
// ===== library types =====

// folder: LIOLink

TYPE "LIOLink_typeDiagnostics"
   STRUCT
      status : Word;   // Status of the Block or error identification when error occurred
      subfunctionStatus : DWord;   // Status or return value of called FB's, FCs and system blocks
      stateNumber : DInt;   // State in the state machine of the block where the error occurred
   END_STRUCT;
END_TYPE

// folder: iJaw

TYPE "UDT_iJawDataRcv"
   STRUCT
      Gauge1 : Word;   // ADC Eingang der Sensorrohdaten (min.: 0 max.: 4096)
      Gauge2 : Word;   // ADC Eingang der Sensorrohdaten (min.: 0 max.: 4096)
      Battery : Byte;   // Rohsignal aktuelle Batteriespannung (min.: 0 .. max.: 157) [V]
      Temperature : Byte;   // Rohsignal Temperatursensor (min.: -40 .. max.: 125) [°C]
      GyroXaxis : Byte;   // Rohsignal Beschleunigungssensor X (min.: -128 .. max.: 127) [g]
      GyroYaxis : Byte;   // Rohsignal Beschleunigungssensor Y (min.: -128 .. max.: 127) [g]
      GyroZaxis : Byte;   // Rohsignal Beschleunigungssensor Z (min.: -128 .. max.: 127) [g]
      Warning : Byte;   // Warnungs-/Fehlercode (Bit0:= Klemmkraft überschritten; Bit1:= Klemmkraft unters
      Force1 : Word;   // Spannkraft Kanal 1 (min.: 0 .. max.: 65,535) [N]
      Force2 : Word;   // Spannkraft Kanal 2 (min.: 0 .. max.: 65,535) [N]
      Reserve1431 : Array[14..31] of Byte;   // Reserve
   END_STRUCT;
END_TYPE

TYPE "UDT_iJawDataSend"
   STRUCT
      nRotSpeedSpindleAct : Int;   // actual rotational speed of the spindle
      pHydCylChamber1Act : Byte;   // actual hydraulic pressure in actuating cylinder chamber for outer clamping
      pHydCylChamber2Act : Byte;   // actual hydraulic pressure in actuating cylinder chamber for outer clamping
      AHydCylChamber1Act : Byte;   // hydraulic area of cylinder chamber for outer clamping
      AHydCylChamber2Act : Byte;   // hydraulic area of cylinder chamber for outer clamping
      Reserve0631 : Array[6..31] of Byte;   // Reserve
   END_STRUCT;
END_TYPE

TYPE "UDT_iJawDataSendUser"
   STRUCT
      xRelCmdSysMode : Bool;   // Trigger send Command change System Mode (see bMode)
      xRelCmdShotOff : Bool;   // Triggr send Command Shut Off
      xRelCmdTara : Bool;   // Trigger send Command Tara
      xReserve1 : Bool;   // Res
      xReserve2 : Bool;   // Res
      xReserve3 : Bool;   // Res
      xReserve4 : Bool;   // Res
      xReserve5 : Bool;   // Res
      bMode : Byte;   // Select Mode (0x1 = continuous mode; 0x2 = state dependent mode
      nRotSpeedSpindleAct : Int;   // actual rotational speed of the spindle
      pHydCylChamber1Act : Byte;   // actual hydraulic pressure in actuating cylinder chamber for outer clamping
      pHydCylChamber2Act : Byte;   // actual hydraulic pressure in actuating cylinder chamber for outer clamping
      AHydCylChamber1Act : Byte;   // hydraulic area of cylinder chamber for outer clamping
      AHydCylChamber2Act : Byte;   // hydraulic area of cylinder chamber for outer clamping
   END_STRUCT;
END_TYPE

TYPE "UDT_iJawDataRcvUser"
   STRUCT
      Gauge1 : UInt;   // ADC Eingang der Sensorrohdaten (min.: 0 max.: 4096)
      Gauge2 : UInt;   // ADC Eingang der Sensorrohdaten (min.: 0 max.: 4096)
      Battery : USInt;   // Rohsignal aktuelle Batteriespannung (min.: 0 .. max.: 157) [V]
      Temperature : SInt;   // Rohsignal Temperatursensor (min.: -40 .. max.: 125) [°C]
      GyroXaxis : SInt;   // Rohsignal Beschleunigungssensor X (min.: -128 .. max.: 127) [g]
      GyroYaxis : SInt;   // Rohsignal Beschleunigungssensor Y (min.: -128 .. max.: 127) [g]
      GyroZaxis : SInt;   // Rohsignal Beschleunigungssensor Z (min.: -128 .. max.: 127) [g]
      Warning : Byte;   // Warnungs-/Fehlercode (Bit0:= Klemmkraft überschritten; Bit1:= Klemmkraft unters
      Force1 : UInt;   // Spannkraft Kanal 1 (min.: 0 .. max.: 65,535) [N]
      Force2 : UInt;   // Spannkraft Kanal 2 (min.: 0 .. max.: 65,535) [N]
      Reserve1431 : Array[14..31] of Byte;   // Reserve
   END_STRUCT;
END_TYPE

// folder: LIOLink/S7-1200/1500/Base blocks

FUNCTION_BLOCK "LIOLink_Device"   // FB50004, SCL
TITLE = LIOLink_Device / LIOLINK_DEVICE
{ S7_Optimized_Access := 'TRUE' }
AUTHOR : SIOS
FAMILY : LIOLink
VERSION : 4.0
// Acyclically reads or writes data records from and to IO-Link devices / Funktionsbaustein zum Lesen und Schreiben von azyklischen Daten auf Geräten mit IO-Link, die auf SIMATIC S7-Steuerungen verwendet werden. (früher IO_LINK_CALL)
   VAR_INPUT
      execute : Bool;   // Request to execute function / Anforderung zum Ausführen der Funktion
      hwID : HW_IO;   // Hardware identifier of IO-Link master module or first sub module / Hardware-Kennung des IO-Link-Mastermoduls (Submodul für ET 200eco PN)
      cap : Int;   // Client Access Point (CAP) 0xB400 or 0x00E3 (227) / Client Access Point (CAP); 0xB400 für ET 200eco PN, CM 8x IO-Link, sonst 0xE003 (227)
      readWrite : Bool;   // FALSE: read-mode, TRUE: write-mode / FALSE: lesen, TRUE: schreiben
      port : Int;   // Port on IO-Link master module / Port am IO-Link-Master-Modul
      index : Int;   // Address parameter index (IO-Link device); 0..32767: IOL-D; 65535: port functions / Adressparameterindex (IO-Link Device); 0..32767: IOL-D; 65535: Portfunktionen
      subindex : Int;   // Address parameter subindex (IO-Link device); 0: full record; 1-255: single parameter / Adressparameter Subindex (IO-Link Device); 0: vollständige Aufzeichnung; 1-255: Einzelparameter
      writeLen : Int;   // Length of writing data (net data); 1..232 / Länge der Schreibdaten (Nettodaten); 1..232
      timeout : Time := T#20S;   // Time after which the request is aborted / Zeit, nach der die Anfrage abgebrochen wird
      pollingPeriod : Time := T#100MS;   // Time period of polling
   END_VAR
   VAR_OUTPUT
      done : Bool;   // TRUE: FB processing successfully completed / TRUE: FB-Bearbeitung erfolgreich abgeschlossen
      busy : Bool;   // TRUE: FB is active and new output values can be expected. / TRUE: FB ist aktiv und neue Ausgangswerte sind zu erwarten.
      error : Bool;   // FALSE: No error / TRUE: An error occurred during the execution of the FB. / FALSE: Kein Fehler / TRUE: Bei der Ausführung des FB ist ein Fehler aufgetreten.
      status : Word := 16#7000;   // 16#0000-16#7FFF: Status of the FB / 16#8000-16#FFFF: Error identification (see following table) / 16#0000-16#7FFF: Status des FB / 16#8000-16#FFFF: Fehleridentifikation (siehe folgende Tabelle)
      diagnostics : "LIOLink_typeDiagnostics";   // Diagnostics information of FB / Diagnoseinformationen der FB
      readLen : Int;   // Length of read data record (number of bytes) / Länge des gelesenen Datensatzes (Anzahl Bytes)
   END_VAR
   VAR_IN_OUT
      record : Array[*] of Byte;   // Data area for reading/writing data (max. 232 byte) / Datenbereich zum Lesen/Schreiben von Daten (max. 232 Byte)
   END_VAR
   VAR
      statExecuteOld : Bool;   // Old value of 'execute' input for edge detection / Alter Wert des 'Execute'-Eingangs für Flankenerkennung
      statDone : Bool;   // Static value for output 'done' / Statischer Wert für Ausgang 'done'
      statBusy : Bool;   // Static value for output 'busy' / Statischer Wert für Ausgang 'besetzt'
      statError : Bool;   // Static value for output 'error' / Statischer Wert für Ausgang 'error'
      statStatus : Word := 16#7000;   // Static value for output 'status' / Statischer Wert für Ausgang 'Status'
      statPollingPeriod : Time := T#100MS;   // Static value for input 'pollingPeriod'
      statHwID : HW_IO;   // Static value for input 'hwID' / Statischer Wert für Eingang 'hwID'
      statHwIDprevious : HW_IO;   // Static value for input 'hwID' from the previous execute / Statischer Wert für Eingang 'hwID'
      statReadWrite : Bool;   // Static value for input 'readWrite' / Stativwert für Eingabe 'readWrite'
      statCap : UInt;   // Static value for input 'cap' / Statischer Wert für Eingabe 'cap'
      statTimeout : Time;   // Static value for input 'timeout' / Statischer Wert für Eingang 'timeout'
      statLen : UInt;   // Length of data to be written to device / Länge der Daten, die auf das Gerät geschrieben werden sollen
      statSubfunctionStatus : DWord;   // Status of WRREC/RDREC or error code from IO-Link Master (%W1: IO-Link Master error, %W0: ISDU error) / Status von WRREC/RDREC oder Fehlercode vom IO-Link-Master (%W1: IO-Link-Master-Fehler, %W0: ISDU-Fehler)
      statFBErrorState : DInt;   // State in the state machine of the block where the error occurred / Zustand in der Zustandsmaschine des Blocks, in dem der Fehler aufgetreten ist
      statFBState : DInt := 0;   // State in the state machine of the FB / Zustand in der Zustandsmaschine der FB
      statEmptyDiagnostics : "LIOLink_typeDiagnostics";   // Empty diagnostics information (for initialization purposes only) / Leere Diagnoseinformationen (nur für Initialisierungszwecke)
      instRdRec : RDREC;   // System function "read data record" / Systemfunktion "Datensatz lesen"
      instWrRec : WRREC;   // System function "write data record" / Systemfunktion "Datensatz schreiben"
      instPoll : TP_TIME;   // poll rate read data record / Abfragerate Datensatz lesen
      instMonitor : TON_TIME;   // request monitoring time / Überwachungszeit anfordern
      statRead : Struct   // data area for reading data / Datenbereich zum Lesen von Daten
         header : Struct   // Header
            call : Struct   // header for read/write data record / Header für Datensatz lesen/schreiben
               extFunctionNum : Byte := 16#08;   // extended function number (fix coded 08h) / erweiterte Funktionsnummer (fix codiert 08h)
               port : Byte;   // variable port (user interface) 0...255 / variabler Port (Benutzeroberfläche) 0...255
               fiIndex : Word := 16#FE4A;   // FI index (fix coded 65098) / FI-Index (fix codiert 65098)
            END_STRUCT;
            iolHeader : Struct   // header for IO-Link / Header für IO-Link
               control : Byte;   // RD_WR = 0 = read = Control:=0x03 / / RD_WR = 1 = write = Control:=0x02 / RD_WR = 0 = lesen = Steuerung:=0x03 / / RD_WR = 1 = schreiben = Steuerung:=0x02
               indexHighByte : Byte;   // index of data record 0…32767 (high byte) / Index des Datensatzes 0…32767 (High Byte)
               indexLowByte : Byte;   // index of data record 0…32767 (low byte) / Index des Datensatzes 0…32767 (Low Byte)
               subindex : Byte;   // subindex for data record 0...255 / Subindex für Datensatz 0...255
            END_STRUCT;
         END_STRUCT;
         data : Array[0..231] of Byte;   // Data
      END_STRUCT;
      statWrite : Struct   // data area for writing data / Datenbereich zum Schreiben von Daten
         header : Struct   // Header
            call : Struct   // header for read/write data record / Header für Datensatz lesen/schreiben
               extFunctionNum : Byte := 16#08;   // extended function number (fix coded 08h) / erweiterte Funktionsnummer (fix codiert 08h)
               port : Byte;   // variable port (user interface) 0...255 / variabler Port (Benutzeroberfläche) 0...255
               fiIndex : Word := 16#FE4A;   // FI index (fix coded 65098) / FI-Index (fix codiert 65098)
            END_STRUCT;
            iolHeader : Struct   // header für IO-Link / Header für IO-Link
               control : Byte;   // RD_WR = 0 = read = Control:=0x03 / / RD_WR = 1 = write = Control:=0x02 / RD_WR = 0 = lesen = Steuerung:=0x03 / / RD_WR = 1 = schreiben = Steuerung:=0x02
               indexHighByte : Byte;   // index of data record 0…32767 (high byte) / Index des Datensatzes 0…32767 (High Byte)
               indexLowByte : Byte;   // index of data record 0…32767 (low byte) / Index des Datensatzes 0…32767 (Low Byte)
               subindex : Byte;   // subindex for data record 0...255 / Subindex für Datensatz 0...255
            END_STRUCT;
         END_STRUCT;
         data : Array[0..231] of Byte;   // Data
      END_STRUCT;
   END_VAR
   VAR_TEMP
      tempExecute : Bool;   // Temporary value for input 'execute' / Temporärer Wert für Eingabe 'execute'
      tempHwID : HW_IO;   // Temporary value for input 'hwID'
      tempPort : Int;   // Temporary value for input 'port'
      tempIndex : Int;   // Temporary value for input 'index'
      tempSubindex : Int;   // Temporary value for input 'subindex'
      tempIndexCounter : DInt;   // run tag for counting loops / Run-Tag für Zählschleifen
   END_VAR
   VAR CONSTANT
      MODE_READ : Bool := FALSE;   // Mode to read data / Modus zum Lesen von Daten
      MODE_WRITE : Bool := TRUE;   // Mode to write data / Modus zum Schreiben von Daten
      MAX_PORT : USInt := 63;   // Max. possible port / max. möglichen Hafen
      MAX_INDEX : UInt := 32767;   // Max. possible index / max. möglicher Index
      INDEX_PORT_FUNC : UInt := 65535;   // Index to address port functions / Index zum Adressieren von Portfunktionen
      MAX_SUBINDEX : USInt := 255;   // Max. possible subindex / max. möglicher Subindex
      MAX_DATA : USInt := 232;   // Max. size of data to be transferred / max. Größe der zu übertragenden Daten
      UPPER_LIMIT : DInt := 231;   // Upper limit of data to be transferred / Obergrenze der zu übertragenden Daten
      FB_STATE_NO_PROCESSING : DInt := 0;   // FB state: No processing / FB-Zustand: Keine Verarbeitung
      FB_STATE_WRITE : DInt := 1;   // FB state: Write data record / Datensatz schreiben
      FB_STATE_POLL : DInt := 2;   // FB state: Wait and poll for response / warten und auf Antwort abfragen
      FB_STATE_READ_CAP : DInt := 3;   // FB state: Read cap / CAP lesen
      IOL_HEADER : UInt := 65098;   // Header IO-Link / Kopfzeile IO-Link
      LEN_HEADER : USInt := 8;   // Length of header / Länge des Headers
      CONTROL_WRITE : Byte := 16#02;   // Write data record / Datensatz schreiben
      CONTROL_READ : Byte := 16#03;   // Read data record / Datensatz lesen
      STATUS_EXECUTION_FINISHED : Word := 16#0000;   // Execution finished without errors / Ausführung ohne Fehler beendet
      STATUS_NO_CALL : Word := 16#7000;   // No job being currently processed / Derzeit wird kein Auftrag bearbeitet
      STATUS_FIRST_CALL : Word := 16#7001;   // First call after incoming new job (rising edge 'execute') / Erster Aufruf nach eingehendem neuen Auftrag (steigende Flanke 'execute')
      STATUS_SUBSEQUENT_CALL : Word := 16#7002;   // Subsequent call during active processing without further details / Nachfolgender Aufruf während aktiver Bearbeitung ohne weitere Angaben
      SUB_STATUS_NO_ERROR : Word := 16#0000;   // No error occured in subfunction call / Fehler: falscher Port
      ERR_WRONG_PORT : Word := 16#8201;   // Error: wrong port / Fehler: falscher Index
      ERR_WRONG_INDEX : Word := 16#8202;   // Error: wrong index / Fehler: falscher Subindex
      ERR_WRONG_SUBINDEX : Word := 16#8203;   // Error: wrong subindex / Fehler: falsche Länge für Datensatz schreiben
      ERR_WRONG_LENGTH : Word := 16#8205;   // Error: wrong length for write data record / Fehler: IO-Link-Master hat Fehlercode zurückgegeben, siehe "Diagnose"
      ERR_IO_LINK : Word := 16#8401;   // Error: IO-Link master returned error code, see "diagnostics" / Fehler: Gelesener Datensatz stimmt nicht mit Anfrage überein
      ERR_INCONSISTENT_DATA : Word := 16#8402;   // Error: Read data record doesn't match request / Fehler: Zeitüberschreitung bei Anforderung
      ERR_REQUEST_TIMEOUT : Word := 16#8403;   // Error: Request timed out / Fehler: Aufgrund eines undefinierten Zustands in der Zustandsmaschine
      ERR_UNDEFINED_STATE : Word := 16#8600;   // Error: due to an undefined state in state machine / Fehler: Aufgrund eines undefinierten Zustands in der Zustandsmaschine
      ERR_WRREC : Word := 16#8601;   // Error: WRREC encountered an error, see "diagnostics" / Fehler: WRREC hat einen Fehler festgestellt, siehe "Diagnose"
      ERR_RDREC : Word := 16#8602;   // Error: RDREC encountered an error, see "diagnostics" / Fehler: RDREC hat einen Fehler festgestellt, siehe "Diagnose"
      STATUS_MASK : DWord := 16#00FF_FF00;   // Mask to filter error codes / Maske zum Filtern von Fehlercodes
      STATUS_RESOURCE_BUSY : DWord := 16#0080_C200;   // Status from WRREC/RDREC: Resource is busy / Status von WRREC/RDREC: Ressource ist beschäftigt
      INDEX_CAP_IOLINK : Word := 16#B000;   // Index of the data record for IOLM_Info. Only IO-Link-Masters with CAP=16#B000 support this call. / Index des Datensatzes für IOLM_Info. Nur IO-Link-Master mit CAP=16#B000 unterstützen diesen Aufruf.
      CAP_LEGACY : Word := 16#00E3;   // Siemens (old) Standard CAP: 227 / Siemens (alt) Standard CAP: 227
      CAP_STANDARD : Word := 16#B400;   // IO-Link Standard CAP: 16#B400 / IO-Link-Standard-CAP: 16#B400
      STATUS_RDREC_VALID : Byte := 16#00;   // Status Code of RDREC in cased of no error occurs
      BITMASK_ERR_RDREC_B3 : Byte := 16#DE;   // Status Code of RDREC in case of an error when reading a data record
      BITMASK_ERR_RDREC_B2 : Byte := 16#80;   // Status Code of RDREC in case of an error when reading a data record - Error according to IEC 61158-6
      BITMASK_ERR_RDREC_B1 : Byte := 16#B0;   // Status Code of RDREC in case of an error when reading a data record - invalid index (cap)
   END_VAR
BEGIN
   REGION BLOCK INFO HEADER
       //===============================================================================
       // Siemens / (c)Copyright 2023
       //-------------------------------------------------------------------------------
       // Title:            LIOLink_Device
       // Function:         Acyclically reads or writes data records from and to IO-Link devices
       // Library:          LIOLink
       // Author:           Siemens Industry Online Support
       // Tested with:      CPU 1513-1 PN FW 2.8
       // Engineering:      TIA Portal V16
       // Restrictions:     S7-1200/1500
       // Requirements:     --
       //-------------------------------------------------------------------------------
       // Change log table:
       // Version  | Date       | Expert in charge       | Changes applied
       //----------|------------|------------------------|------------------------------
       // 02.00.00 | 30.09.2013 | Online Support         | First release for TIA Portal V12 SP1 as IO_LINK_CALL
       // 02.01.00 | 14.03.2014 | Online Support         | Upgrade to TIA Portal V13
       //                                                | Upgrade of system function 'WRREC' from V1.0 to V1.1
       // 03.00.00 | 28.02.2015 | SUP Applications       | Upgrade to TIA Portal V13 SP1
       //                                                | Renamed FB to IO_LINK_DEVICE 
       // 03.01.00 | 15.09.2015 | SUP Applications       | Change of #IOL_INDEX AND #Port lower boundry to 0 and improved behaviour when called in cyclic OBs with > 100 ms
       // 04.00.00 | 01.09.2020 | Online Support         | Implemented Programming styleguide for S7-1200/1500 and PLCopen
       //                                                | Renamed FB to LIOLink_Device 
       // 05.00.00 | 28.02.2023 | SUP SPH                | Added Polling Time as predefined input
       //                                                | #record is changed to a variable array (Array[*])
       //                                                | Changed CAP as predefined variable, added functionality to automatically find CAP of IO-Link-Masters from SIEMENS                                               
       //===============================================================================
   END_REGION

   REGION TRIGGERING
       #tempExecute := #execute; // Work with temporary value / create process image

       IF (#tempExecute = TRUE) AND (#statExecuteOld = FALSE) // Check if FB is triggered
           AND (#statStatus = #STATUS_NO_CALL)
       THEN
           REGION Initialize data
               // First call; initialize FB
               #statDone := FALSE;
               #statBusy := TRUE;
               #statError := FALSE;
               #statStatus := #STATUS_FIRST_CALL;
               #statSubfunctionStatus := #SUB_STATUS_NO_ERROR;
               #statFBErrorState := 0;
               #diagnostics := #statEmptyDiagnostics;
               #readLen := 0;

               // Initialize data area
               #statRead.header."call"."port" := 16#0;
               #statRead.header.iolHeader.indexLowByte := 16#0;
               #statRead.header.iolHeader.indexHighByte := 16#0;
               #statRead.header.iolHeader.subindex := 16#0;
               #tempIndexCounter := 0; // initialize loop counter      
               FOR #tempIndexCounter := 0 TO #UPPER_LIMIT DO
                   #statWrite.data[#tempIndexCounter] := 16#0;
                   #statRead.data[#tempIndexCounter] := 16#0;
               END_FOR;
           END_REGION

           REGION Save inputs
               // Copy input variables to temporary variables
               #tempHwID := #hwID;
               #statReadWrite := #readWrite;
               #statTimeout := #timeout;
               #statPollingPeriod := #pollingPeriod;
               #tempPort := #port;
               #tempIndex := #index;
               #tempSubindex := #subindex;
           END_REGION

           REGION Build header
               // setup call header
               #statWrite.header."call"."port" := INT_TO_BYTE(#tempPort);

               // setup IOL header 
               #statWrite.header.iolHeader.indexLowByte := INT_TO_BYTE(#tempIndex);
               #statWrite.header.iolHeader.indexHighByte := INT_TO_BYTE(SHR(IN := #tempIndex, N := 8));
               #statWrite.header.iolHeader.subindex := INT_TO_BYTE(#tempSubindex);

               // BODY (data max. 232 Byte, Array 0..231 of Byte) 
               IF #statReadWrite = #MODE_WRITE THEN // Write data record requested, copy data from "record"
                   #statWrite.header.iolHeader.control := #CONTROL_WRITE;
                   #statLen := INT_TO_UINT(#writeLen) + #LEN_HEADER; // data length header + data = IO-Link write data record
                   // copy "record" to working area
                   FOR #tempIndexCounter := 0 TO #writeLen - 1 DO
                       #statWrite.data[#tempIndexCounter] := #record[#tempIndexCounter];
                   END_FOR;
               ELSE // Read data record requested
                   // Empty record array
                   FILL_BLK(IN := 16#0,
                            COUNT := #MAX_DATA,
                            OUT => #record[0]);

                   #statWrite.header.iolHeader.control := #CONTROL_READ;
                   #statLen := #LEN_HEADER; // data length only header = IO-Link read data record
               END_IF;
           END_REGION

           REGION Check parameters
               // Check parameters
               IF (#tempPort < 0) OR (#tempPort > #MAX_PORT) THEN
                   #statStatus := #ERR_WRONG_PORT;
               ELSIF (#tempIndex < 0) OR (#tempIndex > #MAX_INDEX AND #tempIndex <> #INDEX_PORT_FUNC) THEN
                   #statStatus := #ERR_WRONG_INDEX;
               ELSIF (#tempSubindex < 0) OR (#tempSubindex > #MAX_SUBINDEX) THEN
                   #statStatus := #ERR_WRONG_SUBINDEX;
               ELSIF #statReadWrite = #MODE_WRITE AND (#writeLen < 1 OR #writeLen > #MAX_DATA) THEN
                   #statStatus := #ERR_WRONG_LENGTH;
               END_IF;
               //save the hwID from the previous execute
               #statHwIDprevious := #statHwID;

               IF #statStatus = #STATUS_FIRST_CALL THEN // Parameters OK
                   IF #cap <> 0 THEN
                       #statCap := INT_TO_UINT(#cap);
                       #statFBState := #FB_STATE_WRITE;
                   ELSIF (#statCap <> WORD_TO_UINT(#CAP_STANDARD) AND #statCap <> WORD_TO_UINT(#CAP_LEGACY)) OR (#statHwIDprevious <> #tempHwID) THEN // check if new device is connected => hwID changed
                       #statFBState := #FB_STATE_READ_CAP;
                   ELSE
                       #statFBState := #FB_STATE_WRITE;
                   END_IF;
               END_IF;
               // save current hwID
               #statHwID := #tempHwID;
           END_REGION

       ELSIF (#statStatus = #STATUS_FIRST_CALL) THEN
           #statStatus := #STATUS_SUBSEQUENT_CALL;
       END_IF;

       // Edge detection 'execute' input
       #statExecuteOld := #tempExecute;
   END_REGION TRIGGERING

   REGION STATE_MACHINE
       CASE #statFBState OF
           #FB_STATE_NO_PROCESSING:
               REGION no processing
                   ; // No processing active
               END_REGION no processing    

           #FB_STATE_READ_CAP:
               REGION get cap
                   // To find out CAP of IO-Link Master, data record with Index 16#B000 is read. If this reading was successful
                   // then CAP is 16#B400 (based on IO-Link Standard). If the reading was not successful and the status of RDREC
                   // is 16#DE80_B0xx, then CAP is 16#00E3 (227, based on Siemens Old Standard for IO-Link Masters).

                   #instRdRec(RECORD := #statRead);

                   IF (#instRdRec.BUSY = FALSE) THEN
                       IF (#instRdRec.VALID = FALSE) AND (#instRdRec.ERROR = FALSE) THEN
                           IF #instRdRec.REQ = FALSE THEN
                               // call read record with Index 16#B000
                               #instRdRec.REQ := true;
                               #instRdRec.ID := #statHwID;
                               #instRdRec.INDEX := WORD_TO_UINT(#INDEX_CAP_IOLINK);
                               #instRdRec.MLEN := 0;
                               #statFBState := #FB_STATE_READ_CAP;
                           END_IF;
                       ELSIF #instRdRec.VALID = TRUE THEN
                           #instRdRec.REQ := FALSE;
                           // if status of RDREC is valid then CAP is 16#B400 (CAP_STANDARD)
                           IF #instRdRec.STATUS.%B3 = #STATUS_RDREC_VALID THEN
                               #statCap := WORD_TO_UINT(#CAP_STANDARD);
                           END_IF;
                           #statFBState := #FB_STATE_WRITE;
                       ELSE
                           // if RDREC is in error state and Status is 16#DE80_B0xx then CAP is 227 (CAP_Legacy)
                           IF (#instRdRec.STATUS.%B3 = #BITMASK_ERR_RDREC_B3) AND (#instRdRec.STATUS.%B2 = #BITMASK_ERR_RDREC_B2) AND (#instRdRec.STATUS.%B1 = #BITMASK_ERR_RDREC_B1) THEN
                               #statCap := WORD_TO_UINT(#CAP_LEGACY);
                               #statFBState := #FB_STATE_WRITE;
                           ELSE
                               #statStatus := #ERR_RDREC;
                               #statSubfunctionStatus := #instRdRec.STATUS;
                               #statCap := 0; //clear CAP if an error occurs
                           END_IF;
                       END_IF;
                   ELSE
                       #instRdRec.REQ := FALSE;
                       IF #instRdRec.ERROR = TRUE THEN
                           #statStatus := #ERR_RDREC;
                           #statSubfunctionStatus := #instRdRec.STATUS;
                           #statCap := 0; //clear CAP if an error occurs
                       END_IF;
                   END_IF;

                   #instRdRec(RECORD := #statRead);
               END_REGION

           #FB_STATE_WRITE:
               REGION write
                   // To read data records, the IO-Link master modules needs to know which port is required. Therefore it is necessary
                   // to send at first a request via write data record (header, 8 byte). As response the IO-Link master module will 
                   // send the required data record.

                   #instWrRec(REQ := TRUE,
                              ID := #statHwID,
                              INDEX := #statCap,
                              LEN := #statLen,
                              RECORD := #statWrite);

                   IF #instWrRec.ERROR THEN
                       IF (#instWrRec.STATUS AND #STATUS_MASK) = #STATUS_RESOURCE_BUSY THEN
                           #instWrRec(REQ := FALSE); // Reset requeset
                       ELSE
                           #statStatus := #ERR_WRREC;
                           #statSubfunctionStatus := #instWrRec.STATUS;
                           #statFBErrorState := #statFBState;
                       END_IF;
                   ELSIF #instWrRec.DONE = TRUE THEN
                       #instWrRec(REQ := FALSE); // Reset requeset

                       #statFBState := #FB_STATE_POLL;
                   END_IF;
               END_REGION write

           #FB_STATE_POLL: // wait and poll for response
               REGION poll
                   #instPoll(IN := TRUE,
                             PT := #statPollingPeriod);

                   // read data record on falling edge
                   #instRdRec(REQ := NOT #instPoll.Q,
                              ID := #statHwID,
                              INDEX := #statCap,
                              MLEN := 0, // read all data available,
                              RECORD := #statRead);

                   IF #instRdRec.ERROR = TRUE THEN
                       IF (#instRdRec.STATUS AND #STATUS_MASK) = #STATUS_RESOURCE_BUSY THEN
                           // Reset requests and try again
                           #instPoll(IN := FALSE,
                                     PT := #statPollingPeriod);

                           #instRdRec(REQ := FALSE,
                                      RECORD := #statRead);
                       ELSE
                           #statStatus := #ERR_RDREC;
                           #statSubfunctionStatus := #instRdRec.STATUS;
                           #statFBErrorState := #statFBState;
                       END_IF;
                   ELSIF #instRdRec.VALID THEN
                       IF // check the response wether it matches the request (compare PORT, INDEX and SUBINDEX)
                           (#statWrite.header."call"."port" <> #statRead.header."call"."port")
                           OR (#statWrite.header.iolHeader.indexHighByte <> #statRead.header.iolHeader.indexHighByte)
                           OR (#statWrite.header.iolHeader.indexLowByte <> #statRead.header.iolHeader.indexLowByte)
                           OR (#statWrite.header.iolHeader.subindex <> #statRead.header.iolHeader.subindex)
                       THEN // read data record doesn't match the request
                           #statStatus := #ERR_INCONSISTENT_DATA;  // output status no consistent data
                       ELSIF #statRead.header.iolHeader.control = B#16#80 THEN // check the response for IO-Link errors
                           // State 0x80 = IOL_CALL_RES PDU shows IO-Link error detect
                           #statStatus := #ERR_IO_LINK;
                           #statSubfunctionStatus.%B3 := #statRead.data[0]; // IO-Link master error code
                           #statSubfunctionStatus.%B2 := #statRead.data[1]; // IO-Link master error code
                           #statSubfunctionStatus.%B1 := #statRead.data[2]; // ISDU error code
                           #statSubfunctionStatus.%B0 := #statRead.data[3]; // ISDU additional code
                           #statFBErrorState := #statFBState;
                       ELSE // read data is valid
                           IF #statReadWrite = #MODE_READ THEN
                               #readLen := UINT_TO_INT(#instRdRec.LEN - #LEN_HEADER);
                               // only data will be output
                               FOR #tempIndexCounter := 0 TO UINT_TO_INT(#instRdRec.LEN - #LEN_HEADER - 1) DO
                                   #record[#tempIndexCounter] := #statRead.data[#tempIndexCounter];
                               END_FOR;
                           END_IF;

                           // Reset requests
                           #instRdRec(REQ := FALSE,
                                      RECORD := #statRead);

                           #instPoll(IN := FALSE,
                                     PT := #statPollingPeriod);

                           #statStatus := #STATUS_EXECUTION_FINISHED;  // request finished
                       END_IF;
                   END_IF;
               END_REGION poll

           ELSE // Undefined state in state machine reached
               REGION undefined state
                   #statStatus := #ERR_UNDEFINED_STATE;
               END_REGION undefined state no relevant case, ready for new request
       END_CASE;
   END_REGION

   REGION MONITORING
       #instMonitor(IN := #statBusy,
                    PT := #statTimeout);

       IF #instMonitor.Q THEN
           #statStatus := #ERR_REQUEST_TIMEOUT; // request time out
       END_IF;
   END_REGION

   REGION OUTPUTS
       // Write outputs
       IF (#statStatus = #STATUS_EXECUTION_FINISHED) AND (#statDone = FALSE) THEN // Execution finished without errors, available only for one cycle
           REGION execution finished
               #statDone := TRUE;
               #statBusy := FALSE;
               #statError := FALSE;
               // execution aborted --> set state no processing
               #statFBState := #FB_STATE_NO_PROCESSING;
           END_REGION execution finished

       ELSIF (#statStatus.%X15 = TRUE) AND (#statError = FALSE) THEN // Error occurred (#statStatus is 16#8000 to 16#FFFF), Error status is true only for one cycle (the second last cycle)
           REGION error occured
               #statDone := FALSE;
               #statBusy := FALSE;
               #statError := TRUE;
               #statCap := 0; //Reset statcap, if error occurs, get cap has to be performed again
               // Write diagnostics
               #diagnostics.status := #statStatus;
               #diagnostics.subfunctionStatus := #statSubfunctionStatus;
               #diagnostics.stateNumber := #statFBErrorState;
               // Call instructions with FALSE to be ready for next job
               #instWrRec(REQ := FALSE);

               #instRdRec(REQ := FALSE,
                          RECORD := #statRead);

               #instPoll(IN := FALSE,
                         PT := #statPollingPeriod);

               // execution aborted --> set state no processing
               #statFBState := #FB_STATE_NO_PROCESSING;
           END_REGION error occured

       ELSIF (#tempExecute = FALSE) AND ((#statDone = TRUE) OR (#statError = TRUE)) THEN // Reset outputs, Last cycle
           REGION execute reset
               #statDone := FALSE;
               #statBusy := FALSE;
               #statError := FALSE;
               #statStatus := #STATUS_NO_CALL;
               #readLen := 0;
           END_REGION execute reset
       END_IF;

       REGION write static values to outputs
           #done := #statDone;
           #busy := #statBusy;
           #error := #statError;
           #status := #statStatus;
           //ENO := NOT #statError;
       END_REGION write static values to outputs
   END_REGION OUTPUTS
END_FUNCTION_BLOCK

// folder: iJaw

FUNCTION_BLOCK "SendRec_iJaw"   // FB3, SCL
{ S7_Optimized_Access := 'TRUE' }
VERSION : 0.1
   VAR_INPUT
      i_LADDR_TigoMaster : HW_DEVICE;
      i_hwIoijaw1 : HW_IO;
      i_hwIoijaw2 : HW_IO;
      i_hwIoijaw3 : HW_IO;
      i_hwIoijaw4 : HW_IO;
      i_hwIoijaw5 : HW_IO;
      i_hwIoijaw6 : HW_IO;
      i_hwIoijaw7 : HW_IO;
      i_hwIoijaw8 : HW_IO;
      i_PN_Act : Bool;
      iJaw_1_vorhanden : Bool;
      iJaw_2_vorhanden : Bool;
      iJaw_3_vorhanden : Bool;
      iJaw_4_vorhanden : Bool;
      iJaw_5_vorhanden : Bool;
      iJaw_6_vorhanden : Bool;
      iJaw_7_vorhanden : Bool;
      iJaw_8_vorhanden : Bool;
      i_CpuRestart : Bool;
      i_Time_PnIoRyd : Time;
      i_UserDaten_iJaw1 : "UDT_iJawDataSendUser";
      i_UserDaten_iJaw2 : "UDT_iJawDataSendUser";
      i_UserDaten_iJaw3 : "UDT_iJawDataSendUser";
      i_UserDaten_iJaw4 : "UDT_iJawDataSendUser";
      i_UserDaten_iJaw5 : "UDT_iJawDataSendUser";
      i_UserDaten_iJaw6 : "UDT_iJawDataSendUser";
      i_UserDaten_iJaw7 : "UDT_iJawDataSendUser";
      i_UserDaten_iJaw8 : "UDT_iJawDataSendUser";
   END_VAR
   VAR_OUTPUT
      o_Error : Bool;
      o_PnTeilAkt : Bool;
      o_UserDaten_iJaw1 : "UDT_iJawDataRcvUser";
      o_UserDaten_iJaw2 : "UDT_iJawDataRcvUser";
      o_UserDaten_iJaw3 : "UDT_iJawDataRcvUser";
      o_UserDaten_iJaw4 : "UDT_iJawDataRcvUser";
      o_UserDaten_iJaw5 : "UDT_iJawDataRcvUser";
      o_UserDaten_iJaw6 : "UDT_iJawDataRcvUser";
      o_UserDaten_iJaw7 : "UDT_iJawDataRcvUser";
      o_UserDaten_iJaw8 : "UDT_iJawDataRcvUser";
   END_VAR
   VAR
      sarrHWIOiJaw : Array[1..#anzahlIjaws] of HW_IO;
      sarrIJawVorhanden : Array[1..#anzahlIjaws] of Bool;
      sx_CpuRestart_old : Bool;
      rcvData : "UDT_iJawDataRcv";
      iRetRcvData : Int;
      iRetSer : Int;
      rcvDaten : Array[1..#laengeRcvDaten] of Byte;
      sarrNcvUserdaten : Array[1..#anzahlIjaws] of "UDT_iJawDataRcvUser";
      sendData : "UDT_iJawDataSend";
      sarrSendUserDaten : Array[1..#anzahlIjaws] of "UDT_iJawDataSendUser";
      iRetSendData : Int;
      instLIOLinkDev : "LIOLink_Device";
      AkuelleSchritt : DInt;
      TON_PNHochlaufzeit : TON_TIME;
      sstrcDeaktAkt : Struct
         ReqAkt : Bool;
         ReqDeak : Bool;
         IstAkt : Bool;
         IstDeak : Bool;
         ModNr : USInt;
         busy : Bool;
         Ret_Val : Int;
         ChangeRequest_old : Bool;
         FP_Changerequest : Bool;
      END_STRUCT;
   END_VAR
   VAR_TEMP
      txAlwaysFalse : Bool;
      txAlwaysTrue : Bool;
      txFPCpuHochlauf : Bool;
      tempI : DInt;
      tempII : DInt;
      tbNull : DInt;
      tempPosSer : DInt;
      tempSchrittNr : DInt;
      tempNschritt : Bool;
      txMin1iJawVorh : Bool;
   END_VAR
   VAR CONSTANT
      anzahlIjaws : DInt := 8;
      laengeRcvDaten : DInt := 33;
      laengeSendDaten : DInt;
      Constant_1 : DInt := 32;
      SCHRITT_1 : DInt := 1;
      SCHRITT_2 : DInt := 2;
   END_VAR
BEGIN
   REGION INIT
       //Bilden Always True und Always False
       #txAlwaysFalse := FALSE;
       #txAlwaysTrue := TRUE;


       //Kopiere HW IO nach Array
       #sarrHWIOiJaw[1] := #i_hwIoijaw1;
       #sarrHWIOiJaw[2] := #i_hwIoijaw2;
       #sarrHWIOiJaw[3] := #i_hwIoijaw3;
       #sarrHWIOiJaw[4] := #i_hwIoijaw4;
       #sarrHWIOiJaw[5] := #i_hwIoijaw5;
       #sarrHWIOiJaw[6] := #i_hwIoijaw6;
       #sarrHWIOiJaw[7] := #i_hwIoijaw7;
       #sarrHWIOiJaw[8] := #i_hwIoijaw8;

       //Kopiere iJaw Vorhanden nach Array
       #sarrIJawVorhanden[1] := #iJaw_1_vorhanden;
       #sarrIJawVorhanden[2] := #iJaw_2_vorhanden;
       #sarrIJawVorhanden[3] := #iJaw_3_vorhanden;
       #sarrIJawVorhanden[4] := #iJaw_4_vorhanden;
       #sarrIJawVorhanden[5] := #iJaw_5_vorhanden;
       #sarrIJawVorhanden[6] := #iJaw_6_vorhanden;
       #sarrIJawVorhanden[7] := #iJaw_7_vorhanden;
       #sarrIJawVorhanden[8] := #iJaw_8_vorhanden;

       //Mindestens 1 iJaw vorhanden
       #txMin1iJawVorh := FALSE;
       FOR #tempI := 1 TO #anzahlIjaws DO
           IF #sarrIJawVorhanden[#tempI] THEN
               #txMin1iJawVorh := TRUE;
               EXIT;
           END_IF;
       END_FOR;

       //Flanke CPU Hochlauf
       IF #txAlwaysTrue AND #i_CpuRestart AND NOT #sx_CpuRestart_old THEN
           #txFPCpuHochlauf := True;
       ELSE
           #txFPCpuHochlauf := False;
       END_IF;
       #sx_CpuRestart_old := #i_CpuRestart;

       //Überbrückung Hochlaufzeit Profinet
       #TON_PNHochlaufzeit(IN := #txAlwaysTrue,
                           PT := #i_Time_PnIoRyd);

   END_REGION
   REGION Daten Init
       //Daten initialisieren
       //Empfangsbereich ablöschen
       FOR #tempI := 1 TO #laengeRcvDaten DO
           #rcvDaten[#tempI] := 0;
       END_FOR;
       //User Empfangsbereich ablöschen
       FOR #tempI := 1 TO #anzahlIjaws DO
           #sarrNcvUserdaten[#tempI].Gauge1 := 0;
           #sarrNcvUserdaten[#tempI].Gauge2 := 0;
           #sarrNcvUserdaten[#tempI].Battery := 0;
           #sarrNcvUserdaten[#tempI].Temperature := 0;
           #sarrNcvUserdaten[#tempI].GyroXaxis := 0;
           #sarrNcvUserdaten[#tempI].GyroYaxis := 0;
           #sarrNcvUserdaten[#tempI].GyroZaxis := 0;
           #sarrNcvUserdaten[#tempI].Warning := 0;
           #sarrNcvUserdaten[#tempI].Force1 := 0;
           #sarrNcvUserdaten[#tempI].Force2 := 0;

           FOR #tempII := 14 TO 31 DO
               #sarrNcvUserdaten[#tempI].Reserve1431[#tempII] := 0;
           END_FOR;

       END_FOR;

       //Sende Daten ablöschen
       #sendData.nRotSpeedSpindleAct := 0;
       #sendData.pHydCylChamber1Act := 0;
       #sendData.pHydCylChamber2Act := 0;
       #sendData.AHydCylChamber1Act := 0;
       #sendData.AHydCylChamber2Act := 0;
       FOR #tempI := 6 TO 31 DO
           #sendData.Reserve0631[#tempI] := 0;
       END_FOR;

       //User Sende Daten ablöschen
       FOR #tempI := 1 TO #anzahlIjaws DO
           #sarrSendUserDaten[#tempI].xRelCmdSysMode := 0;
           #sarrSendUserDaten[#tempI].xRelCmdShotOff := 0;
           #sarrSendUserDaten[#tempI].xRelCmdTara := 0;
           #sarrSendUserDaten[#tempI].xReserve1 := 0;
           #sarrSendUserDaten[#tempI].xReserve2 := 0;
           #sarrSendUserDaten[#tempI].xReserve3 := 0;
           #sarrSendUserDaten[#tempI].xReserve4 := 0;
           #sarrSendUserDaten[#tempI].xReserve5 := 0;
           #sarrSendUserDaten[#tempI].bMode := 0;
           #sarrSendUserDaten[#tempI].nRotSpeedSpindleAct := 0;
           #sarrSendUserDaten[#tempI].pHydCylChamber1Act := 0;
           #sarrSendUserDaten[#tempI].pHydCylChamber2Act := 0;
           #sarrSendUserDaten[#tempI].AHydCylChamber1Act := 0;
           #sarrSendUserDaten[#tempI].AHydCylChamber2Act := 0;

       END_FOR;

   END_REGION

   REGION Profinet Slave aktivieren / deaktivieren
       //Reset bei Hochlauf
       IF #txAlwaysTrue AND #txFPCpuHochlauf THEN
           #sstrcDeaktAkt.ReqAkt := 0;
           #sstrcDeaktAkt.ReqDeak := 0;
           #sstrcDeaktAkt.IstAkt := 0;
           #sstrcDeaktAkt.IstDeak := 0;
           #sstrcDeaktAkt.ModNr := 0;
       END_IF;

       //Request PN Slave aktivieren
       IF #txAlwaysTrue AND #TON_PNHochlaufzeit.Q AND #i_PN_Act AND #txMin1iJawVorh AND NOT #txFPCpuHochlauf AND NOT #sstrcDeaktAkt.IstAkt THEN
           #sstrcDeaktAkt.ModNr := 1;
           #sstrcDeaktAkt.ReqAkt := TRUE;
       END_IF;

       //Request PN Slave deaktivieren
       IF #txAlwaysTrue AND #TON_PNHochlaufzeit.Q AND (NOT #i_PN_Act OR NOT #txMin1iJawVorh) AND NOT #txFPCpuHochlauf AND NOT #sstrcDeaktAkt.IstDeak THEN
           #sstrcDeaktAkt.ModNr := 2;
           #sstrcDeaktAkt.ReqDeak := TRUE;
       END_IF;

       // Setze Bausteinausgang Teilnehmer aktiv
       #o_PnTeilAkt := #txAlwaysTrue AND #sstrcDeaktAkt.IstAkt AND NOT #sstrcDeaktAkt.IstDeak;

       //Teilnehmer aktivieren / deaktivieren
       #sstrcDeaktAkt.Ret_Val := D_ACT_DP(REQ := #sstrcDeaktAkt.ReqAkt OR #sstrcDeaktAkt.ReqDeak, MODE := #sstrcDeaktAkt.ModNr, LADDR := #i_LADDR_TigoMaster, BUSY => #sstrcDeaktAkt.busy);

       //Zustand Aktiviert / deaktiviert speichern
       //Trigger generieren
       IF #sstrcDeaktAkt.Ret_Val = 0 AND #sstrcDeaktAkt.ModNr <> 0 AND NOT #sstrcDeaktAkt.ChangeRequest_old THEN
           #sstrcDeaktAkt.FP_Changerequest := True;
       ELSE
           #sstrcDeaktAkt.FP_Changerequest := false;
       END_IF;
       #sstrcDeaktAkt.ChangeRequest_old := #sstrcDeaktAkt.Ret_Val = 0 AND #sstrcDeaktAkt.ModNr <> 0;

       //Status speicher
       //Slave ist aktiviert
       IF #sstrcDeaktAkt.FP_Changerequest AND #sstrcDeaktAkt.ModNr = 1 THEN
           #sstrcDeaktAkt.ReqAkt := 0;
           #sstrcDeaktAkt.ReqDeak := 0;
           #sstrcDeaktAkt.IstAkt := 1;
           #sstrcDeaktAkt.IstDeak := 0;
           #sstrcDeaktAkt.ModNr := 0;
           //Slave ist deaktiviert
       ELSIF #sstrcDeaktAkt.FP_Changerequest AND #sstrcDeaktAkt.ModNr = 2 THEN
           #sstrcDeaktAkt.ReqAkt := 0;
           #sstrcDeaktAkt.ReqDeak := 0;
           #sstrcDeaktAkt.IstAkt := 0;
           #sstrcDeaktAkt.IstDeak := 1;
           #sstrcDeaktAkt.ModNr := 0;
       END_IF;
   END_REGION
   REGION Daten Empfangen
       //Recive Data from iJaws 1..Anzahl iJaws
       FOR #tempI := 1 TO #anzahlIjaws DO

           //Empfangsbereich ablöschen
           FOR #tempII := 1 TO #laengeRcvDaten DO
               #rcvDaten[#tempII] := 0;
           END_FOR;

           //Daten abholen wenn iJaw N vorhanden
           IF #sstrcDeaktAkt.IstAkt AND #sarrIJawVorhanden[#tempI] THEN
               #iRetRcvData := DPRD_DAT(LADDR := #sarrHWIOiJaw[#tempI], RECORD => #rcvDaten);
           END_IF;

           //Empfangene Daten aufbereiten
           #iRetSer := Deserialize(SRC_ARRAY := #rcvDaten, DEST_VARIABLE => #rcvData, POS := #tempPosSer);

           #sarrNcvUserdaten[#tempI].Gauge1 := WORD_TO_UINT(#rcvData.Gauge1);
           #sarrNcvUserdaten[#tempI].Gauge2 := WORD_TO_UINT(#rcvData.Gauge2);
           #sarrNcvUserdaten[#tempI].Battery := BYTE_TO_USINT(#rcvData.Battery);
           #sarrNcvUserdaten[#tempI].Temperature := BYTE_TO_SINT(#rcvData.Temperature);
           #sarrNcvUserdaten[#tempI].GyroXaxis := BYTE_TO_SINT(#rcvData.GyroXaxis);
           #sarrNcvUserdaten[#tempI].GyroYaxis := BYTE_TO_SINT(#rcvData.GyroYaxis);
           #sarrNcvUserdaten[#tempI].GyroZaxis := BYTE_TO_SINT(#rcvData.GyroZaxis);
           #sarrNcvUserdaten[#tempI].Force1 := WORD_TO_UINT(#rcvData.Force1);
           #sarrNcvUserdaten[#tempI].Force2 := WORD_TO_UINT(#rcvData.Force2);
       END_FOR;

       //Empfangene Daten auf Bausteinausgang schreiben
       #o_UserDaten_iJaw1 := #sarrNcvUserdaten[1];
       #o_UserDaten_iJaw2 := #sarrNcvUserdaten[2];
       #o_UserDaten_iJaw3 := #sarrNcvUserdaten[3];
       #o_UserDaten_iJaw4 := #sarrNcvUserdaten[4];
       #o_UserDaten_iJaw5 := #sarrNcvUserdaten[5];
       #o_UserDaten_iJaw6 := #sarrNcvUserdaten[6];
       #o_UserDaten_iJaw7 := #sarrNcvUserdaten[7];
       #o_UserDaten_iJaw8 := #sarrNcvUserdaten[8];

   END_REGION

   //**************Begin - TODO*******************
   REGION Schrittkette Kommandos schreiben
       // Statement section REGION

   END_REGION
   //**************ENDE - TODO*******************

   REGION Daten senden
       //Daten senden an iJaw 1..Anzahl iJaws

       //Daten ablöschen
       #sendData.nRotSpeedSpindleAct := 0;
       #sendData.pHydCylChamber1Act := 0;
       #sendData.pHydCylChamber2Act := 0;
       #sendData.AHydCylChamber1Act := 0;
       #sendData.AHydCylChamber2Act := 0;
       FOR #tempI := 6 TO 31 DO
           #sendData.Reserve0631[#tempI] := 0;
       END_FOR;

       //Sende Daten vom Bausteineingang einlesen
       #sarrSendUserDaten[1] := #i_UserDaten_iJaw1;
       #sarrSendUserDaten[2] := #i_UserDaten_iJaw2;
       #sarrSendUserDaten[3] := #i_UserDaten_iJaw3;
       #sarrSendUserDaten[4] := #i_UserDaten_iJaw4;
       #sarrSendUserDaten[5] := #i_UserDaten_iJaw5;
       #sarrSendUserDaten[6] := #i_UserDaten_iJaw6;
       #sarrSendUserDaten[7] := #i_UserDaten_iJaw7;
       #sarrSendUserDaten[8] := #i_UserDaten_iJaw8;

       //Daten aufbereiten
       FOR #tempI := 1 TO #anzahlIjaws DO
           //wenn iJaw vorhanden
           IF #sarrIJawVorhanden[#tempI] THEN
               #sendData.nRotSpeedSpindleAct := #sarrSendUserDaten[#tempI].nRotSpeedSpindleAct;
               #sendData.pHydCylChamber1Act := #sarrSendUserDaten[#tempI].pHydCylChamber1Act;
               #sendData.pHydCylChamber2Act := #sarrSendUserDaten[#tempI].pHydCylChamber2Act;
               #sendData.AHydCylChamber1Act := #sarrSendUserDaten[#tempI].AHydCylChamber1Act;
               #sendData.AHydCylChamber2Act := #sarrSendUserDaten[#tempI].AHydCylChamber2Act;

           END_IF;

           //Daten senden
           IF #sstrcDeaktAkt.IstAkt THEN
               #iRetSendData := DPWR_DAT(LADDR := #sarrHWIOiJaw[#tempI], RECORD := #sendData);
           END_IF;
       END_FOR;
   END_REGION
END_FUNCTION_BLOCK

// ===== library: MasterCopy "Kopie von Funktionsbaustein in iJaw" =====

// folder: iJaw

FUNCTION_BLOCK "SendRec_iJaw"   // FB3, SCL
{ S7_Optimized_Access := 'TRUE' }
VERSION : 0.1
   VAR_INPUT
      i_LADDR_TigoMaster : HW_DEVICE;
      i_hwIoijaw1 : HW_IO;
      i_hwIoijaw2 : HW_IO;
      i_hwIoijaw3 : HW_IO;
      i_hwIoijaw4 : HW_IO;
      i_hwIoijaw5 : HW_IO;
      i_hwIoijaw6 : HW_IO;
      i_hwIoijaw7 : HW_IO;
      i_hwIoijaw8 : HW_IO;
      i_PN_Act : Bool;
      iJaw_1_vorhanden : Bool;
      iJaw_2_vorhanden : Bool;
      iJaw_3_vorhanden : Bool;
      iJaw_4_vorhanden : Bool;
      iJaw_5_vorhanden : Bool;
      iJaw_6_vorhanden : Bool;
      iJaw_7_vorhanden : Bool;
      iJaw_8_vorhanden : Bool;
      i_CpuRestart : Bool;
      i_Time_PnIoRyd : Time;
      i_UserDaten_iJaw1 : "UDT_iJawDataSendUser";
      i_UserDaten_iJaw2 : "UDT_iJawDataSendUser";
      i_UserDaten_iJaw3 : "UDT_iJawDataSendUser";
      i_UserDaten_iJaw4 : "UDT_iJawDataSendUser";
      i_UserDaten_iJaw5 : "UDT_iJawDataSendUser";
      i_UserDaten_iJaw6 : "UDT_iJawDataSendUser";
      i_UserDaten_iJaw7 : "UDT_iJawDataSendUser";
      i_UserDaten_iJaw8 : "UDT_iJawDataSendUser";
   END_VAR
   VAR_OUTPUT
      o_Error : Bool;
      o_PnTeilAkt : Bool;
      o_UserDaten_iJaw1 : "UDT_iJawDataRcvUser";
      o_UserDaten_iJaw2 : "UDT_iJawDataRcvUser";
      o_UserDaten_iJaw3 : "UDT_iJawDataRcvUser";
      o_UserDaten_iJaw4 : "UDT_iJawDataRcvUser";
      o_UserDaten_iJaw5 : "UDT_iJawDataRcvUser";
      o_UserDaten_iJaw6 : "UDT_iJawDataRcvUser";
      o_UserDaten_iJaw7 : "UDT_iJawDataRcvUser";
      o_UserDaten_iJaw8 : "UDT_iJawDataRcvUser";
   END_VAR
   VAR
      sarrHWIOiJaw : Array[1..#anzahlIjaws] of HW_IO;
      sarrIJawVorhanden : Array[1..#anzahlIjaws] of Bool;
      sx_CpuRestart_old : Bool;
      rcvData : "UDT_iJawDataRcv";
      iRetRcvData : Int;
      iRetSer : Int;
      rcvDaten : Array[1..#laengeRcvDaten] of Byte;
      sarrNcvUserdaten : Array[1..#anzahlIjaws] of "UDT_iJawDataRcvUser";
      sendData : "UDT_iJawDataSend";
      sarrSendUserDaten : Array[1..#anzahlIjaws] of "UDT_iJawDataSendUser";
      iRetSendData : Int;
      instLIOLinkDev : "LIOLink_Device";
      AkuelleSchritt : DInt;
      TON_PNHochlaufzeit : TON_TIME;
      sstrcDeaktAkt : Struct
         ReqAkt : Bool;
         ReqDeak : Bool;
         IstAkt : Bool;
         IstDeak : Bool;
         ModNr : USInt;
         busy : Bool;
         Ret_Val : Int;
         ChangeRequest_old : Bool;
         FP_Changerequest : Bool;
      END_STRUCT;
   END_VAR
   VAR_TEMP
      txAlwaysFalse : Bool;
      txAlwaysTrue : Bool;
      txFPCpuHochlauf : Bool;
      tempI : DInt;
      tempII : DInt;
      tbNull : DInt;
      tempPosSer : DInt;
      tempSchrittNr : DInt;
      tempNschritt : Bool;
      txMin1iJawVorh : Bool;
   END_VAR
   VAR CONSTANT
      anzahlIjaws : DInt := 8;
      laengeRcvDaten : DInt := 33;
      laengeSendDaten : DInt;
      Constant_1 : DInt := 32;
      SCHRITT_1 : DInt := 1;
      SCHRITT_2 : DInt := 2;
   END_VAR
BEGIN
   REGION INIT
       //Bilden Always True und Always False
       #txAlwaysFalse := FALSE;
       #txAlwaysTrue := TRUE;


       //Kopiere HW IO nach Array
       #sarrHWIOiJaw[1] := #i_hwIoijaw1;
       #sarrHWIOiJaw[2] := #i_hwIoijaw2;
       #sarrHWIOiJaw[3] := #i_hwIoijaw3;
       #sarrHWIOiJaw[4] := #i_hwIoijaw4;
       #sarrHWIOiJaw[5] := #i_hwIoijaw5;
       #sarrHWIOiJaw[6] := #i_hwIoijaw6;
       #sarrHWIOiJaw[7] := #i_hwIoijaw7;
       #sarrHWIOiJaw[8] := #i_hwIoijaw8;

       //Kopiere iJaw Vorhanden nach Array
       #sarrIJawVorhanden[1] := #iJaw_1_vorhanden;
       #sarrIJawVorhanden[2] := #iJaw_2_vorhanden;
       #sarrIJawVorhanden[3] := #iJaw_3_vorhanden;
       #sarrIJawVorhanden[4] := #iJaw_4_vorhanden;
       #sarrIJawVorhanden[5] := #iJaw_5_vorhanden;
       #sarrIJawVorhanden[6] := #iJaw_6_vorhanden;
       #sarrIJawVorhanden[7] := #iJaw_7_vorhanden;
       #sarrIJawVorhanden[8] := #iJaw_8_vorhanden;

       //Mindestens 1 iJaw vorhanden
       #txMin1iJawVorh := FALSE;
       FOR #tempI := 1 TO #anzahlIjaws DO
           IF #sarrIJawVorhanden[#tempI] THEN
               #txMin1iJawVorh := TRUE;
               EXIT;
           END_IF;
       END_FOR;

       //Flanke CPU Hochlauf
       IF #txAlwaysTrue AND #i_CpuRestart AND NOT #sx_CpuRestart_old THEN
           #txFPCpuHochlauf := True;
       ELSE
           #txFPCpuHochlauf := False;
       END_IF;
       #sx_CpuRestart_old := #i_CpuRestart;

       //Überbrückung Hochlaufzeit Profinet
       #TON_PNHochlaufzeit(IN := #txAlwaysTrue,
                           PT := #i_Time_PnIoRyd);

   END_REGION
   REGION Daten Init
       //Daten initialisieren
       //Empfangsbereich ablöschen
       FOR #tempI := 1 TO #laengeRcvDaten DO
           #rcvDaten[#tempI] := 0;
       END_FOR;
       //User Empfangsbereich ablöschen
       FOR #tempI := 1 TO #anzahlIjaws DO
           #sarrNcvUserdaten[#tempI].Gauge1 := 0;
           #sarrNcvUserdaten[#tempI].Gauge2 := 0;
           #sarrNcvUserdaten[#tempI].Battery := 0;
           #sarrNcvUserdaten[#tempI].Temperature := 0;
           #sarrNcvUserdaten[#tempI].GyroXaxis := 0;
           #sarrNcvUserdaten[#tempI].GyroYaxis := 0;
           #sarrNcvUserdaten[#tempI].GyroZaxis := 0;
           #sarrNcvUserdaten[#tempI].Warning := 0;
           #sarrNcvUserdaten[#tempI].Force1 := 0;
           #sarrNcvUserdaten[#tempI].Force2 := 0;

           FOR #tempII := 14 TO 31 DO
               #sarrNcvUserdaten[#tempI].Reserve1431[#tempII] := 0;
           END_FOR;

       END_FOR;

       //Sende Daten ablöschen
       #sendData.nRotSpeedSpindleAct := 0;
       #sendData.pHydCylChamber1Act := 0;
       #sendData.pHydCylChamber2Act := 0;
       #sendData.AHydCylChamber1Act := 0;
       #sendData.AHydCylChamber2Act := 0;
       FOR #tempI := 6 TO 31 DO
           #sendData.Reserve0631[#tempI] := 0;
       END_FOR;

       //User Sende Daten ablöschen
       FOR #tempI := 1 TO #anzahlIjaws DO
           #sarrSendUserDaten[#tempI].xRelCmdSysMode := 0;
           #sarrSendUserDaten[#tempI].xRelCmdShotOff := 0;
           #sarrSendUserDaten[#tempI].xRelCmdTara := 0;
           #sarrSendUserDaten[#tempI].xReserve1 := 0;
           #sarrSendUserDaten[#tempI].xReserve2 := 0;
           #sarrSendUserDaten[#tempI].xReserve3 := 0;
           #sarrSendUserDaten[#tempI].xReserve4 := 0;
           #sarrSendUserDaten[#tempI].xReserve5 := 0;
           #sarrSendUserDaten[#tempI].bMode := 0;
           #sarrSendUserDaten[#tempI].nRotSpeedSpindleAct := 0;
           #sarrSendUserDaten[#tempI].pHydCylChamber1Act := 0;
           #sarrSendUserDaten[#tempI].pHydCylChamber2Act := 0;
           #sarrSendUserDaten[#tempI].AHydCylChamber1Act := 0;
           #sarrSendUserDaten[#tempI].AHydCylChamber2Act := 0;

       END_FOR;

   END_REGION

   REGION Profinet Slave aktivieren / deaktivieren
       //Reset bei Hochlauf
       IF #txAlwaysTrue AND #txFPCpuHochlauf THEN
           #sstrcDeaktAkt.ReqAkt := 0;
           #sstrcDeaktAkt.ReqDeak := 0;
           #sstrcDeaktAkt.IstAkt := 0;
           #sstrcDeaktAkt.IstDeak := 0;
           #sstrcDeaktAkt.ModNr := 0;
       END_IF;

       //Request PN Slave aktivieren
       IF #txAlwaysTrue AND #TON_PNHochlaufzeit.Q AND #i_PN_Act AND #txMin1iJawVorh AND NOT #txFPCpuHochlauf AND NOT #sstrcDeaktAkt.IstAkt THEN
           #sstrcDeaktAkt.ModNr := 1;
           #sstrcDeaktAkt.ReqAkt := TRUE;
       END_IF;

       //Request PN Slave deaktivieren
       IF #txAlwaysTrue AND #TON_PNHochlaufzeit.Q AND (NOT #i_PN_Act OR NOT #txMin1iJawVorh) AND NOT #txFPCpuHochlauf AND NOT #sstrcDeaktAkt.IstDeak THEN
           #sstrcDeaktAkt.ModNr := 2;
           #sstrcDeaktAkt.ReqDeak := TRUE;
       END_IF;

       // Setze Bausteinausgang Teilnehmer aktiv
       #o_PnTeilAkt := #txAlwaysTrue AND #sstrcDeaktAkt.IstAkt AND NOT #sstrcDeaktAkt.IstDeak;

       //Teilnehmer aktivieren / deaktivieren
       #sstrcDeaktAkt.Ret_Val := D_ACT_DP(REQ := #sstrcDeaktAkt.ReqAkt OR #sstrcDeaktAkt.ReqDeak, MODE := #sstrcDeaktAkt.ModNr, LADDR := #i_LADDR_TigoMaster, BUSY => #sstrcDeaktAkt.busy);

       //Zustand Aktiviert / deaktiviert speichern
       //Trigger generieren
       IF #sstrcDeaktAkt.Ret_Val = 0 AND #sstrcDeaktAkt.ModNr <> 0 AND NOT #sstrcDeaktAkt.ChangeRequest_old THEN
           #sstrcDeaktAkt.FP_Changerequest := True;
       ELSE
           #sstrcDeaktAkt.FP_Changerequest := false;
       END_IF;
       #sstrcDeaktAkt.ChangeRequest_old := #sstrcDeaktAkt.Ret_Val = 0 AND #sstrcDeaktAkt.ModNr <> 0;

       //Status speicher
       //Slave ist aktiviert
       IF #sstrcDeaktAkt.FP_Changerequest AND #sstrcDeaktAkt.ModNr = 1 THEN
           #sstrcDeaktAkt.ReqAkt := 0;
           #sstrcDeaktAkt.ReqDeak := 0;
           #sstrcDeaktAkt.IstAkt := 1;
           #sstrcDeaktAkt.IstDeak := 0;
           #sstrcDeaktAkt.ModNr := 0;
           //Slave ist deaktiviert
       ELSIF #sstrcDeaktAkt.FP_Changerequest AND #sstrcDeaktAkt.ModNr = 2 THEN
           #sstrcDeaktAkt.ReqAkt := 0;
           #sstrcDeaktAkt.ReqDeak := 0;
           #sstrcDeaktAkt.IstAkt := 0;
           #sstrcDeaktAkt.IstDeak := 1;
           #sstrcDeaktAkt.ModNr := 0;
       END_IF;
   END_REGION
   REGION Daten Empfangen
       //Recive Data from iJaws 1..Anzahl iJaws
       FOR #tempI := 1 TO #anzahlIjaws DO

           //Empfangsbereich ablöschen
           FOR #tempII := 1 TO #laengeRcvDaten DO
               #rcvDaten[#tempII] := 0;
           END_FOR;

           //Daten abholen wenn iJaw N vorhanden
           IF #sstrcDeaktAkt.IstAkt AND #sarrIJawVorhanden[#tempI] THEN
               #iRetRcvData := DPRD_DAT(LADDR := #sarrHWIOiJaw[#tempI], RECORD => #rcvDaten);
           END_IF;

           //Empfangene Daten aufbereiten
           #iRetSer := Deserialize(SRC_ARRAY := #rcvDaten, DEST_VARIABLE => #rcvData, POS := #tempPosSer);

           #sarrNcvUserdaten[#tempI].Gauge1 := WORD_TO_UINT(#rcvData.Gauge1);
           #sarrNcvUserdaten[#tempI].Gauge2 := WORD_TO_UINT(#rcvData.Gauge2);
           #sarrNcvUserdaten[#tempI].Battery := BYTE_TO_USINT(#rcvData.Battery);
           #sarrNcvUserdaten[#tempI].Temperature := BYTE_TO_SINT(#rcvData.Temperature);
           #sarrNcvUserdaten[#tempI].GyroXaxis := BYTE_TO_SINT(#rcvData.GyroXaxis);
           #sarrNcvUserdaten[#tempI].GyroYaxis := BYTE_TO_SINT(#rcvData.GyroYaxis);
           #sarrNcvUserdaten[#tempI].GyroZaxis := BYTE_TO_SINT(#rcvData.GyroZaxis);
           #sarrNcvUserdaten[#tempI].Force1 := WORD_TO_UINT(#rcvData.Force1);
           #sarrNcvUserdaten[#tempI].Force2 := WORD_TO_UINT(#rcvData.Force2);
       END_FOR;

       //Empfangene Daten auf Bausteinausgang schreiben
       #o_UserDaten_iJaw1 := #sarrNcvUserdaten[1];
       #o_UserDaten_iJaw2 := #sarrNcvUserdaten[2];
       #o_UserDaten_iJaw3 := #sarrNcvUserdaten[3];
       #o_UserDaten_iJaw4 := #sarrNcvUserdaten[4];
       #o_UserDaten_iJaw5 := #sarrNcvUserdaten[5];
       #o_UserDaten_iJaw6 := #sarrNcvUserdaten[6];
       #o_UserDaten_iJaw7 := #sarrNcvUserdaten[7];
       #o_UserDaten_iJaw8 := #sarrNcvUserdaten[8];

   END_REGION

   //**************Begin - TODO*******************
   REGION Schrittkette Kommandos schreiben
       // Statement section REGION

   END_REGION
   //**************ENDE - TODO*******************

   REGION Daten senden
       //Daten senden an iJaw 1..Anzahl iJaws

       //Daten ablöschen
       #sendData.nRotSpeedSpindleAct := 0;
       #sendData.pHydCylChamber1Act := 0;
       #sendData.pHydCylChamber2Act := 0;
       #sendData.AHydCylChamber1Act := 0;
       #sendData.AHydCylChamber2Act := 0;
       FOR #tempI := 6 TO 31 DO
           #sendData.Reserve0631[#tempI] := 0;
       END_FOR;

       //Sende Daten vom Bausteineingang einlesen
       #sarrSendUserDaten[1] := #i_UserDaten_iJaw1;
       #sarrSendUserDaten[2] := #i_UserDaten_iJaw2;
       #sarrSendUserDaten[3] := #i_UserDaten_iJaw3;
       #sarrSendUserDaten[4] := #i_UserDaten_iJaw4;
       #sarrSendUserDaten[5] := #i_UserDaten_iJaw5;
       #sarrSendUserDaten[6] := #i_UserDaten_iJaw6;
       #sarrSendUserDaten[7] := #i_UserDaten_iJaw7;
       #sarrSendUserDaten[8] := #i_UserDaten_iJaw8;

       //Daten aufbereiten
       FOR #tempI := 1 TO #anzahlIjaws DO
           //wenn iJaw vorhanden
           IF #sarrIJawVorhanden[#tempI] THEN
               #sendData.nRotSpeedSpindleAct := #sarrSendUserDaten[#tempI].nRotSpeedSpindleAct;
               #sendData.pHydCylChamber1Act := #sarrSendUserDaten[#tempI].pHydCylChamber1Act;
               #sendData.pHydCylChamber2Act := #sarrSendUserDaten[#tempI].pHydCylChamber2Act;
               #sendData.AHydCylChamber1Act := #sarrSendUserDaten[#tempI].AHydCylChamber1Act;
               #sendData.AHydCylChamber2Act := #sarrSendUserDaten[#tempI].AHydCylChamber2Act;

           END_IF;

           //Daten senden
           IF #sstrcDeaktAkt.IstAkt THEN
               #iRetSendData := DPWR_DAT(LADDR := #sarrHWIOiJaw[#tempI], RECORD := #sendData);
           END_IF;
       END_FOR;
   END_REGION
END_FUNCTION_BLOCK